TYPE "SubAssembly Check_ShW"
VERSION : 0.1
   STRUCT
      Trigger : Bool;
      Result : Int;
      Completed : Bool;
      Q_ID { S7_SetPoint := 'False'} : "SubAssemblyID_ShW";
   END_STRUCT;

END_TYPE

